// TwinCAT 3 PLC project mobject_iot
// Title: mobject-iot
// Company: mobject.io
// Author: mobject dev team
// ProjectVersion: 0.0.0
// ProgramVersion: 3.1.4023.0
// libraries:
//   mobject-core, * (mobject.io)
//   mobject-json, * (mobject.io)
//   Tc2_System, * (Beckhoff Automation GmbH)
//   Tc3_IotBase, * (Beckhoff Automation GmbH)
//   Tc3_Module, * (Beckhoff Automation GmbH)
// project tree:
//   REST/Get/ HttpGet.TcPOU
//   REST/Put/ HttpPut.TcPOU
//   REST/Response/ I_HttpResponse.TcIO
//   _Internal/Response/ HttpResponse.TcPOU

// ---- REST/Response/I_HttpResponse.TcIO
INTERFACE I_HttpResponse EXTENDS I_Disposable

PROPERTY PUBLIC Json : I_JsonPath
GET
END_GET
END_PROPERTY

PROPERTY PUBLIC ResponseCode : udint
GET
END_GET
END_PROPERTY

END_INTERFACE

// ---- REST/Get/HttpGet.TcPOU
{attribute 'linkalways'} 
{attribute 'no_explicit_call' := 'This FB is a CLASS and must be accessed using methods or properties'}
{attribute 'enable_dynamic_creation'}
FUNCTION_BLOCK HttpGet EXTENDS Command
VAR
	url : T_MAXSTRING;
	httpClient : REFERENCE TO FB_IotHttpClient;	
	response : REFERENCE TO I_HttpResponse;
    httpRequest : FB_IotHttpRequest;
END_VAR

METHOD FB_init : BOOL
VAR_INPUT
	bInitRetains : BOOL; // if TRUE, the retain variables are initialized (warm start / cold start)
	bInCopyCode : BOOL;  // if TRUE, the instance afterwards gets moved into the copy code (online change)	
	HttpClient : REFERENCE TO FB_IotHttpClient;
	Url : T_MAXSTRING;
	Response : REFERENCE TO I_HttpResponse;
END_VAR
THIS^.httpClient REF= HttpClient;
THIS^.url := Url;
This^.response ref= Response;
END_METHOD

METHOD PROTECTED OnExecute
VAR_INPUT
	CommandState : I_CommandBusyState;
END_VAR
F_SafeRelease(response);
httpRequest.SendRequest(sUri:= url,fbClient:= httpClient,eRequestType:= ETcIotHttpRequestType.HTTP_GET, 0, 0, 0);
END_METHOD

METHOD PROTECTED WhileBusy
VAR_INPUT
	commandState : I_CommandBusyState;
END_VAR
VAR
	httpResponse : POINTER TO HTTPResponse;
END_VAR
IF httpRequest.bBusy THEN
	 RETURN;
END_IF

IF httpRequest.bError THEN
	commandState.SetError(httpRequest.eErrorId);
	RETURN;
END_IF

httpResponse := __NEW(HttpResponse(HttpRequest := httpRequest));
response := httpResponse^;

commandState.SetDone();
END_METHOD

END_FUNCTION_BLOCK

// ---- _Internal/Response/HttpResponse.TcPOU
{attribute 'linkalways'} 
{attribute 'no_explicit_call' := 'This FB is a CLASS and must be accessed using methods or properties'}
{attribute 'enable_dynamic_creation'}
FUNCTION_BLOCK HttpResponse EXTENDS Disposable IMPLEMENTS I_HttpResponse
VAR
	jsonPath : JsonPath;	
	nStatusCode : UDINT;
	eErrorId : ETcIotHttpRequestError;
	nContentSize : UDINT;
END_VAR

METHOD FB_init : BOOL
VAR_INPUT
	bInitRetains : BOOL; // if TRUE, the retain variables are initialized (warm start / cold start)
	bInCopyCode : BOOL;  // if TRUE, the instance afterwards gets moved into the copy code (online change)
	HttpRequest : REFERENCE TO FB_IotHttpRequest;
END_VAR
nStatusCode := HttpRequest.nStatusCode;
eErrorId := HttpRequest.eErrorId;
nContentSize := HttpRequest.nContentSize;
jsonPath.ParseFromHttpRequest(HttpRequest);
END_METHOD

PROPERTY PUBLIC Json : I_JsonPath
GET
Json := jsonPath;
END_GET
END_PROPERTY

PROPERTY PUBLIC ResponseCode : udint
GET
ResponseCode := nStatusCode;
END_GET
END_PROPERTY

END_FUNCTION_BLOCK

// ---- REST/Put/HttpPut.TcPOU
{attribute 'linkalways'} 
{attribute 'no_explicit_call' := 'This FB is a CLASS and must be accessed using methods or properties'}
{attribute 'enable_dynamic_creation'}
FUNCTION_BLOCK HttpPut EXTENDS Command
VAR
	url : T_MAXSTRING;
	httpClient : REFERENCE TO FB_IotHttpClient;	
	response : REFERENCE TO I_HttpResponse;
    httpRequest : FB_IotHttpRequest;
END_VAR

METHOD FB_init : BOOL
VAR_INPUT
	bInitRetains : BOOL; // if TRUE, the retain variables are initialized (warm start / cold start)
	bInCopyCode : BOOL;  // if TRUE, the instance afterwards gets moved into the copy code (online change)	
	HttpClient : REFERENCE TO FB_IotHttpClient;
	Url : T_MAXSTRING;
	Response : REFERENCE TO I_HttpResponse;
END_VAR
THIS^.httpClient REF= HttpClient;
THIS^.url := Url;
This^.response ref= Response;
END_METHOD

METHOD PROTECTED OnExecute
VAR_INPUT
	CommandState : I_CommandBusyState;
END_VAR
F_SafeRelease(response);
httpRequest.SendRequest(sUri:= url,fbClient:= httpClient,eRequestType:= ETcIotHttpRequestType.HTTP_PUT, 0, 0, 0);
END_METHOD

METHOD PROTECTED WhileBusy
VAR_INPUT
	commandState : I_CommandBusyState;
END_VAR
VAR
	httpResponse : POINTER TO HTTPResponse;
END_VAR
IF httpRequest.bBusy THEN
	 RETURN;
END_IF

IF httpRequest.bError THEN
	commandState.SetError(httpRequest.eErrorId);
	RETURN;
END_IF

httpResponse := __NEW(HttpResponse(HttpRequest := httpRequest));
response := httpResponse^;

commandState.SetDone();
END_METHOD

END_FUNCTION_BLOCK
